    movel([0.070902, -1.350034, -2.596677, -0.765678, 1.570796, 1.641698],accel_mss,speed_ms,0,blend_radius_m)
    movel([0.072260, -1.349314, -2.597153, -0.765922, 1.570796, 1.643056],accel_mss,speed_ms,0,blend_radius_m)
    movel([0.073070, -1.348013, -2.598010, -0.766365, 1.570796, 1.643866],accel_mss,speed_ms,0,blend_radius_m)
    movel([0.072836, -1.347012, -2.598669, -0.766708, 1.570796, 1.643632],accel_mss,speed_ms,0,blend_radius_m)
    movel([0.071683, -1.346767, -2.598830, -0.766792, 1.570796, 1.642479],accel_mss,speed_ms,0,blend_radius_m)
    movel([0.071683, -1.324561, -2.588363, -0.799465, 1.570796, 1.642479],accel_mss,speed_ms,0,blend_radius_m)
    movel([0.085049, -1.312983, -2.595633, -0.803774, 1.570796, 1.655845],accel_mss,speed_ms,0,blend_radius_m)
    movel([0.085049, -1.335367, -2.606227, -0.770796, 1.570796, 1.655845],accel_mss,speed_ms,0,blend_radius_m)
    movel([0.085444, -1.331348, -2.608792, -0.772249, 1.570796, 1.656240],accel_mss,speed_ms,0,blend_radius_m)
    movel([0.084179, -1.331324, -2.608807, -0.772258, 1.570796, 1.654975],accel_mss,speed_ms,0,blend_radius_m)
    movel([0.083165, -1.330827, -2.609122, -0.772439, 1.570796, 1.653962],accel_mss,speed_ms,0,blend_radius_m)
    movel([0.082588, -1.329954, -2.609676, -0.772759, 1.570796, 1.653384],accel_mss,speed_ms,0,blend_radius_m)
    movel([0.082504, -1.328932, -2.610323, -0.773134, 1.570796, 1.653300],accel_mss,speed_ms,0,blend_radius_m)
    movel([0.083255, -1.326914, -2.611596, -0.773878, 1.570796, 1.654051],accel_mss,speed_ms,0,blend_radius_m)
    movel([0.084328, -1.325638, -2.612398, -0.774352, 1.570796, 1.655124],accel_mss,speed_ms,0,blend_radius_m)
    movel([0.085303, -1.324858, -2.612888, -0.774643, 1.570796, 1.656099],accel_mss,speed_ms,0,blend_radius_m)
    movel([0.086132, -1.324375, -2.613190, -0.774823, 1.570796, 1.656928],accel_mss,speed_ms,0,blend_radius_m)
    movel([0.086527, -1.320394, -2.615673, -0.776322, 1.570796, 1.657323],accel_mss,speed_ms,0,blend_radius_m)
    movel([0.088109, -1.319882, -2.615990, -0.776517, 1.570796, 1.658906],accel_mss,speed_ms,0,blend_radius_m)
    movel([0.087707, -1.323869, -2.613507, -0.775013, 1.570796, 1.658503],accel_mss,speed_ms,0,blend_radius_m)
    movel([0.089323, -1.323988, -2.613433, -0.774968, 1.570796, 1.660119],accel_mss,speed_ms,0,blend_radius_m)
    movel([0.090412, -1.324915, -2.612853, -0.774622, 1.570796, 1.661208],accel_mss,speed_ms,0,blend_radius_m)
    movel([0.090641, -1.326329, -2.611965, -0.774096, 1.570796, 1.661438],accel_mss,speed_ms,0,blend_radius_m)
    movel([0.090159, -1.327852, -2.611005, -0.773532, 1.570796, 1.660955],accel_mss,speed_ms,0,blend_radius_m)
    movel([0.088700, -1.329704, -2.609835, -0.772850, 1.570796, 1.659496],accel_mss,speed_ms,0,blend_radius_m)
    movel([0.087006, -1.330851, -2.609108, -0.772431, 1.570796, 1.657802],accel_mss,speed_ms,0,blend_radius_m)
    movel([0.086604, -1.334875, -2.606542, -0.770972, 1.570796, 1.657400],accel_mss,speed_ms,0,blend_radius_m)
    movel([0.085049, -1.335367, -2.606227, -0.770796, 1.570796, 1.655845],accel_mss,speed_ms,0,blend_radius_m)
    movel([0.085444, -1.331348, -2.608792, -0.772249, 1.570796, 1.656240],accel_mss,speed_ms,0,blend_radius_m)
    movel([0.084179, -1.331324, -2.608807, -0.772258, 1.570796, 1.654975],accel_mss,speed_ms,0,blend_radius_m)
    movel([0.083165, -1.330827, -2.609122, -0.772439, 1.570796, 1.653962],accel_mss,speed_ms,0,blend_radius_m)
    movel([0.082588, -1.329954, -2.609676, -0.772759, 1.570796, 1.653384],accel_mss,speed_ms,0,blend_radius_m)
    movel([0.082504, -1.328932, -2.610323, -0.773134, 1.570796, 1.653300],accel_mss,speed_ms,0,blend_radius_m)
    movel([0.083255, -1.326914, -2.611596, -0.773878, 1.570796, 1.654051],accel_mss,speed_ms,0,blend_radius_m)
    movel([0.084328, -1.325638, -2.612398, -0.774352, 1.570796, 1.655124],accel_mss,speed_ms,0,blend_radius_m)
    movel([0.085303, -1.324858, -2.612888, -0.774643, 1.570796, 1.656099],accel_mss,speed_ms,0,blend_radius_m)
    movel([0.086132, -1.324375, -2.613190, -0.774823, 1.570796, 1.656928],accel_mss,speed_ms,0,blend_radius_m)
    movel([0.086527, -1.320394, -2.615673, -0.776322, 1.570796, 1.657323],accel_mss,speed_ms,0,blend_radius_m)
    movel([0.088109, -1.319882, -2.615990, -0.776517, 1.570796, 1.658906],accel_mss,speed_ms,0,blend_radius_m)
    movel([0.087707, -1.323869, -2.613507, -0.775013, 1.570796, 1.658503],accel_mss,speed_ms,0,blend_radius_m)
    movel([0.089323, -1.323988, -2.613433, -0.774968, 1.570796, 1.660119],accel_mss,speed_ms,0,blend_radius_m)
    movel([0.090412, -1.324915, -2.612853, -0.774622, 1.570796, 1.661208],accel_mss,speed_ms,0,blend_radius_m)
    movel([0.090641, -1.326329, -2.611965, -0.774096, 1.570796, 1.661438],accel_mss,speed_ms,0,blend_radius_m)
    movel([0.090159, -1.327852, -2.611005, -0.773532, 1.570796, 1.660955],accel_mss,speed_ms,0,blend_radius_m)
    movel([0.088700, -1.329704, -2.609835, -0.772850, 1.570796, 1.659496],accel_mss,speed_ms,0,blend_radius_m)
    movel([0.087006, -1.330851, -2.609108, -0.772431, 1.570796, 1.657802],accel_mss,speed_ms,0,blend_radius_m)
    movel([0.086604, -1.334875, -2.606542, -0.770972, 1.570796, 1.657400],accel_mss,speed_ms,0,blend_radius_m)
    movel([0.085049, -1.335367, -2.606227, -0.770796, 1.570796, 1.655845],accel_mss,speed_ms,0,blend_radius_m)
    movel([0.085049, -1.312983, -2.595633, -0.803774, 1.570796, 1.655845],accel_mss,speed_ms,0,blend_radius_m)
    movel([0.074252, -1.294457, -2.606902, -0.811029, 1.570796, 1.645049],accel_mss,speed_ms,0,blend_radius_m)
    movel([0.074252, -1.317114, -2.617702, -0.777573, 1.570796, 1.645049],accel_mss,speed_ms,0,blend_radius_m)
    movel([0.075203, -1.317104, -2.617708, -0.777577, 1.570796, 1.646000],accel_mss,speed_ms,0,blend_radius_m)
    movel([0.075659, -1.317927, -2.617200, -0.777262, 1.570796, 1.646456],accel_mss,speed_ms,0,blend_radius_m)
    movel([0.075058, -1.319090, -2.616481, -0.776818, 1.570796, 1.645854],accel_mss,speed_ms,0,blend_radius_m)
    movel([0.074027, -1.319755, -2.616069, -0.776565, 1.570796, 1.644823],accel_mss,speed_ms,0,blend_radius_m)
    movel([0.055660, -1.326016, -2.612161, -0.774212, 1.570796, 1.626456],accel_mss,speed_ms,0,blend_radius_m)
    movel([0.054684, -1.326038, -2.612147, -0.774203, 1.570796, 1.625481],accel_mss,speed_ms,0,blend_radius_m)
    movel([0.054234, -1.325244, -2.612646, -0.774499, 1.570796, 1.625031],accel_mss,speed_ms,0,blend_radius_m)
    movel([0.054836, -1.324070, -2.613381, -0.774937, 1.570796, 1.625633],accel_mss,speed_ms,0,blend_radius_m)
    movel([0.055828, -1.323418, -2.613789, -0.775182, 1.570796, 1.626625],accel_mss,speed_ms,0,blend_radius_m)
    movel([0.054836, -1.324070, -2.613381, -0.774937, 1.570796, 1.625633],accel_mss,speed_ms,0,blend_radius_m)
    movel([0.054234, -1.325244, -2.612646, -0.774499, 1.570796, 1.625031],accel_mss,speed_ms,0,blend_radius_m)
    movel([0.054684, -1.326038, -2.612147, -0.774203, 1.570796, 1.625481],accel_mss,speed_ms,0,blend_radius_m)
    movel([0.055660, -1.326016, -2.612161, -0.774212, 1.570796, 1.626456],accel_mss,speed_ms,0,blend_radius_m)
    movel([0.074027, -1.319755, -2.616069, -0.776565, 1.570796, 1.644823],accel_mss,speed_ms,0,blend_radius_m)
    movel([0.075058, -1.319090, -2.616481, -0.776818, 1.570796, 1.645854],accel_mss,speed_ms,0,blend_radius_m)
    movel([0.075659, -1.317927, -2.617200, -0.777262, 1.570796, 1.646456],accel_mss,speed_ms,0,blend_radius_m)
    movel([0.075203, -1.317104, -2.617708, -0.777577, 1.570796, 1.646000],accel_mss,speed_ms,0,blend_radius_m)
    movel([0.074252, -1.317114, -2.617702, -0.777573, 1.570796, 1.645049],accel_mss,speed_ms,0,blend_radius_m)
    movel([0.074252, -1.294457, -2.606902, -0.811029, 1.570796, 1.645049],accel_mss,speed_ms,0,blend_radius_m)
    movel([0.056123, -1.285439, -2.612231, -0.814720, 1.570796, 1.626919],accel_mss,speed_ms,0,blend_radius_m)
    movel([0.056123, -1.308222, -2.623130, -0.781036, 1.570796, 1.626919],accel_mss,speed_ms,0,blend_radius_m)
    movel([0.055744, -1.308276, -2.623098, -0.781015, 1.570796, 1.626540],accel_mss,speed_ms,0,blend_radius_m)
    movel([0.056123, -1.308222, -2.623130, -0.781036, 1.570796, 1.626919],accel_mss,speed_ms,0,blend_radius_m)
    movel([0.056123, -1.285439, -2.612231, -0.814720, 1.570796, 1.626919],accel_mss,speed_ms,0,blend_radius_m)
    movel([0.055744, -1.285493, -2.612198, -0.814697, 1.570796, 1.626540],accel_mss,speed_ms,0,blend_radius_m)
    movel([0.055744, -1.308276, -2.623098, -0.781015, 1.570796, 1.626540],accel_mss,speed_ms,0,blend_radius_m)
    movel([0.055431, -1.308121, -2.623192, -0.781076, 1.570796, 1.626227],accel_mss,speed_ms,0,blend_radius_m)
    movel([0.055343, -1.307815, -2.623376, -0.781197, 1.570796, 1.626139],accel_mss,speed_ms,0,blend_radius_m)
    movel([0.055975, -1.297990, -2.629249, -0.785150, 1.570796, 1.626772],accel_mss,speed_ms,0,blend_radius_m)
    movel([0.056126, -1.297559, -2.629504, -0.785326, 1.570796, 1.626922],accel_mss,speed_ms,0,blend_radius_m)
    movel([0.056534, -1.297139, -2.629752, -0.785498, 1.570796, 1.627330],accel_mss,speed_ms,0,blend_radius_m)
    movel([0.056857, -1.296975, -2.629849, -0.785565, 1.570796, 1.627654],accel_mss,speed_ms,0,blend_radius_m)
    movel([0.065790, -1.293762, -2.631738, -0.786889, 1.570796, 1.636586],accel_mss,speed_ms,0,blend_radius_m)
    movel([0.066189, -1.293703, -2.631772, -0.786914, 1.570796, 1.636985],accel_mss,speed_ms,0,blend_radius_m)
    movel([0.066524, -1.293939, -2.631634, -0.786816, 1.570796, 1.637320],accel_mss,speed_ms,0,blend_radius_m)
    movel([0.066573, -1.294183, -2.631491, -0.786715, 1.570796, 1.637370],accel_mss,speed_ms,0,blend_radius_m)
    movel([0.065818, -1.304106, -2.625608, -0.782675, 1.570796, 1.636615],accel_mss,speed_ms,0,blend_radius_m)
    movel([0.065712, -1.304447, -2.625404, -0.782538, 1.570796, 1.636508],accel_mss,speed_ms,0,blend_radius_m)
    movel([0.065160, -1.305003, -2.625070, -0.782316, 1.570796, 1.635956],accel_mss,speed_ms,0,blend_radius_m)
    movel([0.056123, -1.308222, -2.623130, -0.781036, 1.570796, 1.626919],accel_mss,speed_ms,0,blend_radius_m)
    movel([0.055744, -1.308276, -2.623098, -0.781015, 1.570796, 1.626540],accel_mss,speed_ms,0,blend_radius_m)
    movel([0.055431, -1.308121, -2.623192, -0.781076, 1.570796, 1.626227],accel_mss,speed_ms,0,blend_radius_m)
    movel([0.055343, -1.307815, -2.623376, -0.781197, 1.570796, 1.626139],accel_mss,speed_ms,0,blend_radius_m)
    movel([0.055975, -1.297990, -2.629249, -0.785150, 1.570796, 1.626772],accel_mss,speed_ms,0,blend_radius_m)
    movel([0.056126, -1.297559, -2.629504, -0.785326, 1.570796, 1.626922],accel_mss,speed_ms,0,blend_radius_m)
    movel([0.056534, -1.297139, -2.629752, -0.785498, 1.570796, 1.627330],accel_mss,speed_ms,0,blend_radius_m)
    movel([0.056857, -1.296975, -2.629849, -0.785565, 1.570796, 1.627654],accel_mss,speed_ms,0,blend_radius_m)
    movel([0.065790, -1.293762, -2.631738, -0.786889, 1.570796, 1.636586],accel_mss,speed_ms,0,blend_radius_m)
    movel([0.066189, -1.293703, -2.631772, -0.786914, 1.570796, 1.636985],accel_mss,speed_ms,0,blend_radius_m)
    movel([0.066524, -1.293939, -2.631634, -0.786816, 1.570796, 1.637320],accel_mss,speed_ms,0,blend_radius_m)
    movel([0.066573, -1.294183, -2.631491, -0.786715, 1.570796, 1.637370],accel_mss,speed_ms,0,blend_radius_m)
    movel([0.065818, -1.304106, -2.625608, -0.782675, 1.570796, 1.636615],accel_mss,speed_ms,0,blend_radius_m)
    movel([0.065712, -1.304447, -2.625404, -0.782538, 1.570796, 1.636508],accel_mss,speed_ms,0,blend_radius_m)
    movel([0.065160, -1.305003, -2.625070, -0.782316, 1.570796, 1.635956],accel_mss,speed_ms,0,blend_radius_m)
    movel([0.056123, -1.308222, -2.623130, -0.781036, 1.570796, 1.626919],accel_mss,speed_ms,0,blend_radius_m)
    movel([0.055744, -1.308276, -2.623098, -0.781015, 1.570796, 1.626540],accel_mss,speed_ms,0,blend_radius_m)
    movel([0.055744, -1.285493, -2.612198, -0.814697, 1.570796, 1.626540],accel_mss,speed_ms,0,blend_radius_m)
    movel([0.066316, -1.281088, -2.614764, -0.816537, 1.570796, 1.637112],accel_mss,speed_ms,0,blend_radius_m)
    movel([0.066316, -1.303932, -2.625713, -0.782745, 1.570796, 1.637112],accel_mss,speed_ms,0,blend_radius_m)
    movel([0.067077, -1.294004, -2.631596, -0.786789, 1.570796, 1.637873],accel_mss,speed_ms,0,blend_radius_m)
    movel([0.067232, -1.293569, -2.631851, -0.786969, 1.570796, 1.638029],accel_mss,speed_ms,0,blend_radius_m)
    movel([0.067632, -1.293153, -2.632094, -0.787141, 1.570796, 1.638428],accel_mss,speed_ms,0,blend_radius_m)
    movel([0.067957, -1.292990, -2.632190, -0.787209, 1.570796, 1.638754],accel_mss,speed_ms,0,blend_radius_m)
    movel([0.076939, -1.289824, -2.634035, -0.788530, 1.570796, 1.647735],accel_mss,speed_ms,0,blend_radius_m)
    movel([0.077324, -1.289773, -2.634065, -0.788551, 1.570796, 1.648120],accel_mss,speed_ms,0,blend_radius_m)
    movel([0.077670, -1.290011, -2.633927, -0.788452, 1.570796, 1.648467],accel_mss,speed_ms,0,blend_radius_m)
    movel([0.077702, -1.290262, -2.633781, -0.788346, 1.570796, 1.648499],accel_mss,speed_ms,0,blend_radius_m)
    movel([0.076817, -1.300287, -2.627887, -0.784214, 1.570796, 1.647614],accel_mss,speed_ms,0,blend_radius_m)
    movel([0.076706, -1.300631, -2.627683, -0.784075, 1.570796, 1.647503],accel_mss,speed_ms,0,blend_radius_m)
    movel([0.076147, -1.301188, -2.627352, -0.783850, 1.570796, 1.646944],accel_mss,speed_ms,0,blend_radius_m)
    movel([0.067076, -1.304355, -2.625459, -0.782575, 1.570796, 1.637872],accel_mss,speed_ms,0,blend_radius_m)
    movel([0.066696, -1.304406, -2.625428, -0.782554, 1.570796, 1.637492],accel_mss,speed_ms,0,blend_radius_m)
    movel([0.066386, -1.304246, -2.625524, -0.782619, 1.570796, 1.637182],accel_mss,speed_ms,0,blend_radius_m)
    movel([0.066316, -1.303932, -2.625713, -0.782745, 1.570796, 1.637112],accel_mss,speed_ms,0,blend_radius_m)
    movel([0.067077, -1.294004, -2.631596, -0.786789, 1.570796, 1.637873],accel_mss,speed_ms,0,blend_radius_m)
    movel([0.067232, -1.293569, -2.631851, -0.786969, 1.570796, 1.638029],accel_mss,speed_ms,0,blend_radius_m)
    movel([0.067632, -1.293153, -2.632094, -0.787141, 1.570796, 1.638428],accel_mss,speed_ms,0,blend_radius_m)
    movel([0.067957, -1.292990, -2.632190, -0.787209, 1.570796, 1.638754],accel_mss,speed_ms,0,blend_radius_m)
    movel([0.076939, -1.289824, -2.634035, -0.788530, 1.570796, 1.647735],accel_mss,speed_ms,0,blend_radius_m)
    movel([0.077324, -1.289773, -2.634065, -0.788551, 1.570796, 1.648120],accel_mss,speed_ms,0,blend_radius_m)
    movel([0.077670, -1.290011, -2.633927, -0.788452, 1.570796, 1.648467],accel_mss,speed_ms,0,blend_radius_m)
    movel([0.077702, -1.290262, -2.633781, -0.788346, 1.570796, 1.648499],accel_mss,speed_ms,0,blend_radius_m)
    movel([0.076817, -1.300287, -2.627887, -0.784214, 1.570796, 1.647614],accel_mss,speed_ms,0,blend_radius_m)
    movel([0.076706, -1.300631, -2.627683, -0.784075, 1.570796, 1.647503],accel_mss,speed_ms,0,blend_radius_m)
    movel([0.076147, -1.301188, -2.627352, -0.783850, 1.570796, 1.646944],accel_mss,speed_ms,0,blend_radius_m)
    movel([0.067076, -1.304355, -2.625459, -0.782575, 1.570796, 1.637872],accel_mss,speed_ms,0,blend_radius_m)
    movel([0.066696, -1.304406, -2.625428, -0.782554, 1.570796, 1.637492],accel_mss,speed_ms,0,blend_radius_m)
    movel([0.066386, -1.304246, -2.625524, -0.782619, 1.570796, 1.637182],accel_mss,speed_ms,0,blend_radius_m)
    movel([0.066316, -1.303932, -2.625713, -0.782745, 1.570796, 1.637112],accel_mss,speed_ms,0,blend_radius_m)
    movel([0.066316, -1.281088, -2.614764, -0.816537, 1.570796, 1.637112],accel_mss,speed_ms,0,blend_radius_m)
    movel([0.077699, -1.271769, -2.620113, -0.820507, 1.570796, 1.648495],accel_mss,speed_ms,0,blend_radius_m)
    movel([0.077699, -1.294738, -2.631165, -0.786486, 1.570796, 1.648495],accel_mss,speed_ms,0,blend_radius_m)
    movel([0.078051, -1.293512, -2.631884, -0.786993, 1.570796, 1.648848],accel_mss,speed_ms,0,blend_radius_m)
    movel([0.079104, -1.292040, -2.632745, -0.787604, 1.570796, 1.649901],accel_mss,speed_ms,0,blend_radius_m)
    movel([0.080305, -1.291064, -2.633314, -0.788011, 1.570796, 1.651101],accel_mss,speed_ms,0,blend_radius_m)
    movel([0.081398, -1.290544, -2.633617, -0.788229, 1.570796, 1.652194],accel_mss,speed_ms,0,blend_radius_m)
    movel([0.143384, -1.270405, -2.645076, -0.796908, 1.570796, 1.714180],accel_mss,speed_ms,0,blend_radius_m)
    movel([0.144886, -1.270259, -2.645157, -0.796973, 1.570796, 1.715682],accel_mss,speed_ms,0,blend_radius_m)
    movel([0.146370, -1.271729, -2.644338, -0.796322, 1.570796, 1.717167],accel_mss,speed_ms,0,blend_radius_m)
    movel([0.146362, -1.272534, -2.643888, -0.795966, 1.570796, 1.717158],accel_mss,speed_ms,0,blend_radius_m)
    movel([0.136356, -1.335897, -2.605886, -0.770605, 1.570796, 1.707152],accel_mss,speed_ms,0,blend_radius_m)
    movel([0.135447, -1.337785, -2.604673, -0.769931, 1.570796, 1.706243],accel_mss,speed_ms,0,blend_radius_m)
    movel([0.133630, -1.339278, -2.603709, -0.769402, 1.570796, 1.704426],accel_mss,speed_ms,0,blend_radius_m)
    movel([0.132691, -1.339647, -2.603471, -0.769272, 1.570796, 1.703488],accel_mss,speed_ms,0,blend_radius_m)
    movel([0.075442, -1.356489, -2.592380, -0.763520, 1.570796, 1.646238],accel_mss,speed_ms,0,blend_radius_m)
    movel([0.074761, -1.356638, -2.592280, -0.763471, 1.570796, 1.645557],accel_mss,speed_ms,0,blend_radius_m)
    movel([0.072688, -1.355806, -2.592837, -0.763746, 1.570796, 1.643484],accel_mss,speed_ms,0,blend_radius_m)
    movel([0.072498, -1.354758, -2.593538, -0.764093, 1.570796, 1.643295],accel_mss,speed_ms,0,blend_radius_m)
    movel([0.077699, -1.294738, -2.631165, -0.786486, 1.570796, 1.648495],accel_mss,speed_ms,0,blend_radius_m)
    movel([0.078051, -1.293512, -2.631884, -0.786993, 1.570796, 1.648848],accel_mss,speed_ms,0,blend_radius_m)
    movel([0.079104, -1.292040, -2.632745, -0.787604, 1.570796, 1.649901],accel_mss,speed_ms,0,blend_radius_m)
    movel([0.080305, -1.291064, -2.633314, -0.788011, 1.570796, 1.651101],accel_mss,speed_ms,0,blend_radius_m)
    movel([0.081398, -1.290544, -2.633617, -0.788229, 1.570796, 1.652194],accel_mss,speed_ms,0,blend_radius_m)
    movel([0.143384, -1.270405, -2.645076, -0.796908, 1.570796, 1.714180],accel_mss,speed_ms,0,blend_radius_m)
    movel([0.144886, -1.270259, -2.645157, -0.796973, 1.570796, 1.715682],accel_mss,speed_ms,0,blend_radius_m)
    movel([0.146370, -1.271729, -2.644338, -0.796322, 1.570796, 1.717167],accel_mss,speed_ms,0,blend_radius_m)
    movel([0.146362, -1.272534, -2.643888, -0.795966, 1.570796, 1.717158],accel_mss,speed_ms,0,blend_radius_m)
    movel([0.136356, -1.335897, -2.605886, -0.770605, 1.570796, 1.707152],accel_mss,speed_ms,0,blend_radius_m)
    movel([0.135447, -1.337785, -2.604673, -0.769931, 1.570796, 1.706243],accel_mss,speed_ms,0,blend_radius_m)
    movel([0.133630, -1.339278, -2.603709, -0.769402, 1.570796, 1.704426],accel_mss,speed_ms,0,blend_radius_m)
    movel([0.132691, -1.339647, -2.603471, -0.769272, 1.570796, 1.703488],accel_mss,speed_ms,0,blend_radius_m)
    movel([0.075442, -1.356489, -2.592380, -0.763520, 1.570796, 1.646238],accel_mss,speed_ms,0,blend_radius_m)
    movel([0.074761, -1.356638, -2.592280, -0.763471, 1.570796, 1.645557],accel_mss,speed_ms,0,blend_radius_m)
    movel([0.072688, -1.355806, -2.592837, -0.763746, 1.570796, 1.643484],accel_mss,speed_ms,0,blend_radius_m)
    movel([0.072498, -1.354758, -2.593538, -0.764093, 1.570796, 1.643295],accel_mss,speed_ms,0,blend_radius_m)
    movel([0.077699, -1.294738, -2.631165, -0.786486, 1.570796, 1.648495],accel_mss,speed_ms,0,blend_radius_m)
    movel([0.077699, -1.271769, -2.620113, -0.820507, 1.570796, 1.648495],accel_mss,speed_ms,0,blend_radius_m)
    movel([0.087111, -1.280077, -2.615350, -0.816962, 1.570796, 1.657907],accel_mss,speed_ms,0,blend_radius_m)
    movel([0.087111, -1.302935, -2.626309, -0.783145, 1.570796, 1.657907],accel_mss,speed_ms,0,blend_radius_m)
    movel([0.089943, -1.301594, -2.627110, -0.783685, 1.570796, 1.660740],accel_mss,speed_ms,0,blend_radius_m)
    movel([0.092948, -1.301071, -2.627421, -0.783897, 1.570796, 1.663745],accel_mss,speed_ms,0,blend_radius_m)
    movel([0.095895, -1.301822, -2.626974, -0.783593, 1.570796, 1.666691],accel_mss,speed_ms,0,blend_radius_m)
    movel([0.097574, -1.303847, -2.625763, -0.782778, 1.570796, 1.668370],accel_mss,speed_ms,0,blend_radius_m)
    movel([0.097857, -1.306436, -2.624208, -0.781745, 1.570796, 1.668653],accel_mss,speed_ms,0,blend_radius_m)
    movel([0.096894, -1.309520, -2.622345, -0.780525, 1.570796, 1.667690],accel_mss,speed_ms,0,blend_radius_m)
    movel([0.094719, -1.312655, -2.620437, -0.779297, 1.570796, 1.665515],accel_mss,speed_ms,0,blend_radius_m)
    movel([0.091120, -1.315592, -2.618638, -0.778159, 1.570796, 1.661916],accel_mss,speed_ms,0,blend_radius_m)
    movel([0.088391, -1.316831, -2.617876, -0.777682, 1.570796, 1.659188],accel_mss,speed_ms,0,blend_radius_m)
    movel([0.084693, -1.317301, -2.617586, -0.777502, 1.570796, 1.655489],accel_mss,speed_ms,0,blend_radius_m)
    movel([0.082521, -1.316624, -2.618003, -0.777761, 1.570796, 1.653318],accel_mss,speed_ms,0,blend_radius_m)
    movel([0.081191, -1.315361, -2.618780, -0.778248, 1.570796, 1.651987],accel_mss,speed_ms,0,blend_radius_m)
    movel([0.080499, -1.312129, -2.620758, -0.779502, 1.570796, 1.651296],accel_mss,speed_ms,0,blend_radius_m)
    movel([0.081621, -1.308623, -2.622888, -0.780878, 1.570796, 1.652418],accel_mss,speed_ms,0,blend_radius_m)
    movel([0.083541, -1.305906, -2.624527, -0.781955, 1.570796, 1.654337],accel_mss,speed_ms,0,blend_radius_m)
    movel([0.087111, -1.302935, -2.626309, -0.783145, 1.570796, 1.657907],accel_mss,speed_ms,0,blend_radius_m)
    movel([0.089943, -1.301594, -2.627110, -0.783685, 1.570796, 1.660740],accel_mss,speed_ms,0,blend_radius_m)
    movel([0.092948, -1.301071, -2.627421, -0.783897, 1.570796, 1.663745],accel_mss,speed_ms,0,blend_radius_m)
    movel([0.095895, -1.301822, -2.626974, -0.783593, 1.570796, 1.666691],accel_mss,speed_ms,0,blend_radius_m)
    movel([0.097574, -1.303847, -2.625763, -0.782778, 1.570796, 1.668370],accel_mss,speed_ms,0,blend_radius_m)
    movel([0.097857, -1.306436, -2.624208, -0.781745, 1.570796, 1.668653],accel_mss,speed_ms,0,blend_radius_m)
    movel([0.096894, -1.309520, -2.622345, -0.780525, 1.570796, 1.667690],accel_mss,speed_ms,0,blend_radius_m)
    movel([0.094719, -1.312655, -2.620437, -0.779297, 1.570796, 1.665515],accel_mss,speed_ms,0,blend_radius_m)
    movel([0.091120, -1.315592, -2.618638, -0.778159, 1.570796, 1.661916],accel_mss,speed_ms,0,blend_radius_m)
    movel([0.088391, -1.316831, -2.617876, -0.777682, 1.570796, 1.659188],accel_mss,speed_ms,0,blend_radius_m)
    movel([0.084693, -1.317301, -2.617586, -0.777502, 1.570796, 1.655489],accel_mss,speed_ms,0,blend_radius_m)
    movel([0.082521, -1.316624, -2.618003, -0.777761, 1.570796, 1.653318],accel_mss,speed_ms,0,blend_radius_m)
    movel([0.081191, -1.315361, -2.618780, -0.778248, 1.570796, 1.651987],accel_mss,speed_ms,0,blend_radius_m)
    movel([0.080499, -1.312129, -2.620758, -0.779502, 1.570796, 1.651296],accel_mss,speed_ms,0,blend_radius_m)
    movel([0.081621, -1.308623, -2.622888, -0.780878, 1.570796, 1.652418],accel_mss,speed_ms,0,blend_radius_m)
    movel([0.083541, -1.305906, -2.624527, -0.781955, 1.570796, 1.654337],accel_mss,speed_ms,0,blend_radius_m)
    movel([0.087111, -1.302935, -2.626309, -0.783145, 1.570796, 1.657907],accel_mss,speed_ms,0,blend_radius_m)
    movel([0.087111, -1.280077, -2.615350, -0.816962, 1.570796, 1.657907],accel_mss,speed_ms,0,blend_radius_m)
    movel([0.074534, -1.291116, -2.608888, -0.812385, 1.570796, 1.645331],accel_mss,speed_ms,0,blend_radius_m)
    movel([0.074534, -1.313820, -2.619725, -0.778844, 1.570796, 1.645331],accel_mss,speed_ms,0,blend_radius_m)
    movel([0.075490, -1.313797, -2.619739, -0.778853, 1.570796, 1.646286],accel_mss,speed_ms,0,blend_radius_m)
    movel([0.075946, -1.314635, -2.619226, -0.778528, 1.570796, 1.646743],accel_mss,speed_ms,0,blend_radius_m)
    movel([0.075342, -1.315805, -2.618507, -0.778077, 1.570796, 1.646139],accel_mss,speed_ms,0,blend_radius_m)
    movel([0.074307, -1.316475, -2.618095, -0.777819, 1.570796, 1.645103],accel_mss,speed_ms,0,blend_radius_m)
    movel([0.055869, -1.322790, -2.614181, -0.775418, 1.570796, 1.626665],accel_mss,speed_ms,0,blend_radius_m)
    movel([0.054890, -1.322813, -2.614167, -0.775409, 1.570796, 1.625686],accel_mss,speed_ms,0,blend_radius_m)
    movel([0.054438, -1.322016, -2.614664, -0.775709, 1.570796, 1.625235],accel_mss,speed_ms,0,blend_radius_m)
    movel([0.055044, -1.320824, -2.615405, -0.776159, 1.570796, 1.625840],accel_mss,speed_ms,0,blend_radius_m)
    movel([0.056039, -1.320179, -2.615806, -0.776404, 1.570796, 1.626835],accel_mss,speed_ms,0,blend_radius_m)
    movel([0.055044, -1.320824, -2.615405, -0.776159, 1.570796, 1.625840],accel_mss,speed_ms,0,blend_radius_m)
    movel([0.054438, -1.322016, -2.614664, -0.775709, 1.570796, 1.625235],accel_mss,speed_ms,0,blend_radius_m)
    movel([0.054890, -1.322813, -2.614167, -0.775409, 1.570796, 1.625686],accel_mss,speed_ms,0,blend_radius_m)
    movel([0.055869, -1.322790, -2.614181, -0.775418, 1.570796, 1.626665],accel_mss,speed_ms,0,blend_radius_m)
    movel([0.074307, -1.316475, -2.618095, -0.777819, 1.570796, 1.645103],accel_mss,speed_ms,0,blend_radius_m)
    movel([0.075342, -1.315805, -2.618507, -0.778077, 1.570796, 1.646139],accel_mss,speed_ms,0,blend_radius_m)
    movel([0.075946, -1.314635, -2.619226, -0.778528, 1.570796, 1.646743],accel_mss,speed_ms,0,blend_radius_m)
    movel([0.075490, -1.313797, -2.619739, -0.778853, 1.570796, 1.646286],accel_mss,speed_ms,0,blend_radius_m)
    movel([0.074534, -1.313820, -2.619725, -0.778844, 1.570796, 1.645331],accel_mss,speed_ms,0,blend_radius_m)
    movel([0.074534, -1.291116, -2.608888, -0.812385, 1.570796, 1.645331],accel_mss,speed_ms,0,blend_radius_m)
    movel([0.078136, -1.266790, -2.622927, -0.822672, 1.570796, 1.648932],accel_mss,speed_ms,0,blend_radius_m)
    movel([0.078136, -1.289824, -2.634035, -0.788530, 1.570796, 1.648932],accel_mss,speed_ms,0,blend_radius_m)
    movel([0.081088, -1.257101, -2.652369, -0.802919, 1.570796, 1.651884],accel_mss,speed_ms,0,blend_radius_m)
    movel([0.115247, -1.244981, -2.658826, -0.808581, 1.570796, 1.686044],accel_mss,speed_ms,0,blend_radius_m)
    movel([0.110999, -1.278720, -2.640406, -0.793262, 1.570796, 1.681795],accel_mss,speed_ms,0,blend_radius_m)
    movel([0.078136, -1.289824, -2.634035, -0.788530, 1.570796, 1.648932],accel_mss,speed_ms,0,blend_radius_m)
    movel([0.081088, -1.257101, -2.652369, -0.802919, 1.570796, 1.651884],accel_mss,speed_ms,0,blend_radius_m)
    movel([0.115247, -1.244981, -2.658826, -0.808581, 1.570796, 1.686044],accel_mss,speed_ms,0,blend_radius_m)
    movel([0.110999, -1.278720, -2.640406, -0.793262, 1.570796, 1.681795],accel_mss,speed_ms,0,blend_radius_m)
    movel([0.078136, -1.289824, -2.634035, -0.788530, 1.570796, 1.648932],accel_mss,speed_ms,0,blend_radius_m)
    movel([0.078136, -1.266790, -2.622927, -0.822672, 1.570796, 1.648932],accel_mss,speed_ms,0,blend_radius_m)
    movel([0.083617, -1.231766, -2.641880, -0.838743, 1.570796, 1.654413],accel_mss,speed_ms,0,blend_radius_m)
    movel([0.083617, -1.255223, -2.653381, -0.803785, 1.570796, 1.654413],accel_mss,speed_ms,0,blend_radius_m)
    movel([0.081966, -1.255223, -2.653381, -0.803785, 1.570796, 1.652762],accel_mss,speed_ms,0,blend_radius_m)
    movel([0.081377, -1.253942, -2.654069, -0.804378, 1.570796, 1.652173],accel_mss,speed_ms,0,blend_radius_m)
    movel([0.082222, -1.252143, -2.655032, -0.805214, 1.570796, 1.653018],accel_mss,speed_ms,0,blend_radius_m)
    movel([0.084027, -1.250873, -2.655709, -0.805807, 1.570796, 1.654823],accel_mss,speed_ms,0,blend_radius_m)
    movel([0.113133, -1.240460, -2.661190, -0.810739, 1.570796, 1.683929],accel_mss,speed_ms,0,blend_radius_m)
    movel([0.115154, -1.240390, -2.661227, -0.810773, 1.570796, 1.685950],accel_mss,speed_ms,0,blend_radius_m)
    movel([0.115667, -1.241693, -2.660548, -0.810148, 1.570796, 1.686463],accel_mss,speed_ms,0,blend_radius_m)
    movel([0.114721, -1.243574, -2.659565, -0.809251, 1.570796, 1.685518],accel_mss,speed_ms,0,blend_radius_m)
    movel([0.112914, -1.244813, -2.658915, -0.808661, 1.570796, 1.683710],accel_mss,speed_ms,0,blend_radius_m)
    movel([0.083617, -1.255223, -2.653381, -0.803785, 1.570796, 1.654413],accel_mss,speed_ms,0,blend_radius_m)
    movel([0.081966, -1.255223, -2.653381, -0.803785, 1.570796, 1.652762],accel_mss,speed_ms,0,blend_radius_m)
    movel([0.081377, -1.253942, -2.654069, -0.804378, 1.570796, 1.652173],accel_mss,speed_ms,0,blend_radius_m)
    movel([0.082222, -1.252143, -2.655032, -0.805214, 1.570796, 1.653018],accel_mss,speed_ms,0,blend_radius_m)
    movel([0.084027, -1.250873, -2.655709, -0.805807, 1.570796, 1.654823],accel_mss,speed_ms,0,blend_radius_m)
    movel([0.113133, -1.240460, -2.661190, -0.810739, 1.570796, 1.683929],accel_mss,speed_ms,0,blend_radius_m)
    movel([0.115154, -1.240390, -2.661227, -0.810773, 1.570796, 1.685950],accel_mss,speed_ms,0,blend_radius_m)
    movel([0.115667, -1.241693, -2.660548, -0.810148, 1.570796, 1.686463],accel_mss,speed_ms,0,blend_radius_m)
    movel([0.114721, -1.243574, -2.659565, -0.809251, 1.570796, 1.685518],accel_mss,speed_ms,0,blend_radius_m)
    movel([0.112914, -1.244813, -2.658915, -0.808661, 1.570796, 1.683710],accel_mss,speed_ms,0,blend_radius_m)
    movel([0.083617, -1.255223, -2.653381, -0.803785, 1.570796, 1.654413],accel_mss,speed_ms,0,blend_radius_m)
    movel([0.083617, -1.231766, -2.641880, -0.838743, 1.570796, 1.654413],accel_mss,speed_ms,0,blend_radius_m)
    movel([0.084119, -1.226373, -2.644671, -0.841345, 1.570796, 1.654916],accel_mss,speed_ms,0,blend_radius_m)
    movel([0.084119, -1.249889, -2.656233, -0.806267, 1.570796, 1.654916],accel_mss,speed_ms,0,blend_radius_m)
    movel([0.082460, -1.249880, -2.656238, -0.806271, 1.570796, 1.653256],accel_mss,speed_ms,0,blend_radius_m)
    movel([0.081867, -1.248603, -2.656915, -0.806871, 1.570796, 1.652663],accel_mss,speed_ms,0,blend_radius_m)
    movel([0.082718, -1.246788, -2.657875, -0.807726, 1.570796, 1.653514],accel_mss,speed_ms,0,blend_radius_m)
    movel([0.084534, -1.245503, -2.658552, -0.808334, 1.570796, 1.655331],accel_mss,speed_ms,0,blend_radius_m)
    movel([0.113824, -1.234941, -2.664043, -0.813405, 1.570796, 1.684620],accel_mss,speed_ms,0,blend_radius_m)
    movel([0.115857, -1.234865, -2.664082, -0.813442, 1.570796, 1.686654],accel_mss,speed_ms,0,blend_radius_m)
    movel([0.116373, -1.236178, -2.663407, -0.812804, 1.570796, 1.687169],accel_mss,speed_ms,0,blend_radius_m)
    movel([0.115421, -1.238063, -2.662433, -0.811892, 1.570796, 1.686218],accel_mss,speed_ms,0,blend_radius_m)
    movel([0.113601, -1.239330, -2.661777, -0.811282, 1.570796, 1.684397],accel_mss,speed_ms,0,blend_radius_m)
    movel([0.084119, -1.249889, -2.656233, -0.806267, 1.570796, 1.654916],accel_mss,speed_ms,0,blend_radius_m)
    movel([0.082460, -1.249880, -2.656238, -0.806271, 1.570796, 1.653256],accel_mss,speed_ms,0,blend_radius_m)
    movel([0.081867, -1.248603, -2.656915, -0.806871, 1.570796, 1.652663],accel_mss,speed_ms,0,blend_radius_m)
    movel([0.082718, -1.246788, -2.657875, -0.807726, 1.570796, 1.653514],accel_mss,speed_ms,0,blend_radius_m)
    movel([0.084534, -1.245503, -2.658552, -0.808334, 1.570796, 1.655331],accel_mss,speed_ms,0,blend_radius_m)
    movel([0.113824, -1.234941, -2.664043, -0.813405, 1.570796, 1.684620],accel_mss,speed_ms,0,blend_radius_m)
    movel([0.115857, -1.234865, -2.664082, -0.813442, 1.570796, 1.686654],accel_mss,speed_ms,0,blend_radius_m)
    movel([0.116373, -1.236178, -2.663407, -0.812804, 1.570796, 1.687169],accel_mss,speed_ms,0,blend_radius_m)
    movel([0.115421, -1.238063, -2.662433, -0.811892, 1.570796, 1.686218],accel_mss,speed_ms,0,blend_radius_m)
    movel([0.113601, -1.239330, -2.661777, -0.811282, 1.570796, 1.684397],accel_mss,speed_ms,0,blend_radius_m)
    movel([0.084119, -1.249889, -2.656233, -0.806267, 1.570796, 1.654916],accel_mss,speed_ms,0,blend_radius_m)
    movel([0.084119, -1.226373, -2.644671, -0.841345, 1.570796, 1.654916],accel_mss,speed_ms,0,blend_radius_m)
    movel([0.082158, -1.221877, -2.646972, -0.843540, 1.570796, 1.652954],accel_mss,speed_ms,0,blend_radius_m)
    movel([0.082158, -1.245441, -2.658584, -0.808363, 1.570796, 1.652954],accel_mss,speed_ms,0,blend_radius_m)
    movel([0.084426, -1.221050, -2.671067, -0.820273, 1.570796, 1.655223],accel_mss,speed_ms,0,blend_radius_m)
    movel([0.120058, -1.207711, -2.677603, -0.827074, 1.570796, 1.690855],accel_mss,speed_ms,0,blend_radius_m)
    movel([0.116788, -1.232939, -2.665069, -0.814381, 1.570796, 1.687585],accel_mss,speed_ms,0,blend_radius_m)
    movel([0.082158, -1.245441, -2.658584, -0.808363, 1.570796, 1.652954],accel_mss,speed_ms,0,blend_radius_m)
    movel([0.084426, -1.221050, -2.671067, -0.820273, 1.570796, 1.655223],accel_mss,speed_ms,0,blend_radius_m)
    movel([0.120058, -1.207711, -2.677603, -0.827074, 1.570796, 1.690855],accel_mss,speed_ms,0,blend_radius_m)
    movel([0.116788, -1.232939, -2.665069, -0.814381, 1.570796, 1.687585],accel_mss,speed_ms,0,blend_radius_m)
    movel([0.082158, -1.245441, -2.658584, -0.808363, 1.570796, 1.652954],accel_mss,speed_ms,0,blend_radius_m)
    movel([0.082158, -1.221877, -2.646972, -0.843540, 1.570796, 1.652954],accel_mss,speed_ms,0,blend_radius_m)
    movel([0.087478, -1.194133, -2.660671, -0.857585, 1.570796, 1.658274],accel_mss,speed_ms,0,blend_radius_m)
    movel([0.087478, -1.217967, -2.672595, -0.821827, 1.570796, 1.658274],accel_mss,speed_ms,0,blend_radius_m)
    movel([0.086755, -1.218152, -2.672504, -0.821733, 1.570796, 1.657551],accel_mss,speed_ms,0,blend_radius_m)
    movel([0.085053, -1.217509, -2.672821, -0.822059, 1.570796, 1.655849],accel_mss,speed_ms,0,blend_radius_m)
    movel([0.084857, -1.216468, -2.673334, -0.822586, 1.570796, 1.655653],accel_mss,speed_ms,0,blend_radius_m)
    movel([0.085826, -1.206213, -2.678325, -0.827851, 1.570796, 1.656622],accel_mss,speed_ms,0,blend_radius_m)
    movel([0.086062, -1.205296, -2.678766, -0.828328, 1.570796, 1.656858],accel_mss,speed_ms,0,blend_radius_m)
    movel([0.087792, -1.203110, -2.679812, -0.829467, 1.570796, 1.658589],accel_mss,speed_ms,0,blend_radius_m)
    movel([0.088994, -1.202420, -2.680141, -0.829828, 1.570796, 1.659790],accel_mss,speed_ms,0,blend_radius_m)
    movel([0.119490, -1.190705, -2.685650, -0.836034, 1.570796, 1.690286],accel_mss,speed_ms,0,blend_radius_m)
    movel([0.120724, -1.190507, -2.685742, -0.836140, 1.570796, 1.691521],accel_mss,speed_ms,0,blend_radius_m)
    movel([0.122064, -1.191655, -2.685209, -0.835525, 1.570796, 1.692861],accel_mss,speed_ms,0,blend_radius_m)
    movel([0.122078, -1.192342, -2.684889, -0.835158, 1.570796, 1.692874],accel_mss,speed_ms,0,blend_radius_m)
    movel([0.120679, -1.202968, -2.679880, -0.829542, 1.570796, 1.691476],accel_mss,speed_ms,0,blend_radius_m)
    movel([0.120290, -1.204144, -2.679318, -0.828928, 1.570796, 1.691086],accel_mss,speed_ms,0,blend_radius_m)
    movel([0.118762, -1.205950, -2.678451, -0.827988, 1.570796, 1.689558],accel_mss,speed_ms,0,blend_radius_m)
    movel([0.117429, -1.206722, -2.678080, -0.827587, 1.570796, 1.688225],accel_mss,speed_ms,0,blend_radius_m)
    movel([0.087478, -1.217967, -2.672595, -0.821827, 1.570796, 1.658274],accel_mss,speed_ms,0,blend_radius_m)
    movel([0.086755, -1.218152, -2.672504, -0.821733, 1.570796, 1.657551],accel_mss,speed_ms,0,blend_radius_m)
    movel([0.085053, -1.217509, -2.672821, -0.822059, 1.570796, 1.655849],accel_mss,speed_ms,0,blend_radius_m)
    movel([0.084857, -1.216468, -2.673334, -0.822586, 1.570796, 1.655653],accel_mss,speed_ms,0,blend_radius_m)
    movel([0.085826, -1.206213, -2.678325, -0.827851, 1.570796, 1.656622],accel_mss,speed_ms,0,blend_radius_m)
    movel([0.086062, -1.205296, -2.678766, -0.828328, 1.570796, 1.656858],accel_mss,speed_ms,0,blend_radius_m)
    movel([0.087792, -1.203110, -2.679812, -0.829467, 1.570796, 1.658589],accel_mss,speed_ms,0,blend_radius_m)
    movel([0.088994, -1.202420, -2.680141, -0.829828, 1.570796, 1.659790],accel_mss,speed_ms,0,blend_radius_m)
    movel([0.119490, -1.190705, -2.685650, -0.836034, 1.570796, 1.690286],accel_mss,speed_ms,0,blend_radius_m)
    movel([0.120724, -1.190507, -2.685742, -0.836140, 1.570796, 1.691521],accel_mss,speed_ms,0,blend_radius_m)
    movel([0.122064, -1.191655, -2.685209, -0.835525, 1.570796, 1.692861],accel_mss,speed_ms,0,blend_radius_m)
    movel([0.122078, -1.192342, -2.684889, -0.835158, 1.570796, 1.692874],accel_mss,speed_ms,0,blend_radius_m)
    movel([0.120679, -1.202968, -2.679880, -0.829542, 1.570796, 1.691476],accel_mss,speed_ms,0,blend_radius_m)
    movel([0.120290, -1.204144, -2.679318, -0.828928, 1.570796, 1.691086],accel_mss,speed_ms,0,blend_radius_m)
    movel([0.118762, -1.205950, -2.678451, -0.827988, 1.570796, 1.689558],accel_mss,speed_ms,0,blend_radius_m)
    movel([0.117429, -1.206722, -2.678080, -0.827587, 1.570796, 1.688225],accel_mss,speed_ms,0,blend_radius_m)
    movel([0.087478, -1.217967, -2.672595, -0.821827, 1.570796, 1.658274],accel_mss,speed_ms,0,blend_radius_m)
    movel([0.087478, -1.112936, -2.609802, -0.989651, 1.570796, 1.658274],accel_mss,speed_ms,0,blend_radius_m)
    # End of main program
  end

  Machining3()
end
